TYPE MaterialSlot :
STRUCT
	material : STRING;
	occupied AT %I* : BOOL;
END_STRUCT
END_TYPE

(* stored: Version 1.1.0.1, ProductVersion 3.1.4024.11
   DUT MaterialSlot: Id {3fe1af31-012a-4c8b-89b1-4b54a3455f56} *)
